FUNCTION_BLOCK PsdChuck EXTENDS ChuckBase
VAR_INPUT
	IoChuckPsd : IoChuckPsd;
END_VAR
VAR_OUTPUT
END_VAR
VAR
	{attribute 'OPC.UA.DA' := '0'}
	_config : PsdChuckConfig;
	
	{attribute 'OPC.UA.DA' := '0'}
	_deliverMessages : INT;
	
	WaferPresenceMsg : STRING(255);
	
	{attribute 'OPC.UA.DA' := '0'}
	_initDevice : BOOL;
	
	{attribute 'OPC.UA.DA' := '0'}
	_itemInit : INT;
	
	{attribute 'OPC.UA.DA' := '0'}
	_itemScheduler : INT;
	{attribute 'OPC.UA.DA' := '0'}
	_itemRaisedProperties : INT;
	{attribute 'OPC.UA.DA' := '0'}
	_pulseGenerator : TON;
	
	{region 'Commands'}
		
	{attribute 'OPC.UA.DA' := '0'}			  		   
	_raisePropertiesCmd : BOOL;
			
	{endregion}	
		
	{attribute 'OPC.UA.DA' := '0'}
	message : STRING;
	{attribute 'OPC.UA.DA' := '0'}
	_waferPresenceSensorCounter : UINT;
		 
END_VAR

SUPER^();

// Init device
InitDevice(); 

// Deliver messages
CASE _deliverMessages OF		
	EFeedbackMsgPsdChuck.WaferPresenceMsg :
		WaferPresenceMsg := message;		
END_CASE
	
_deliverMessages := 0;

// Commands	
RaisePropertiesChanged(_raisePropertiesCmd);

IF (NOT _raisePropertiesCmd) THEN
	MessageScheduler();
END_IF

METHOD FB_init : BOOL
VAR_INPUT
	bInitRetains : BOOL; // if TRUE, the retain variables are initialized (warm start / cold start)
	bInCopyCode : BOOL;  // if TRUE, the instance afterwards gets moved into the copy code (online change)
	Config : PsdChuckConfig;
END_VAR
IF Config.IsEnabled THEN
	_config := Config;
	
	SUPER^._chuckConfig.Name := Config.Name;
	SUPER^._chuckConfig.DeviceID := Config.DeviceID;
	SUPER^._chuckConfig.IsEnabled := Config.IsEnabled;
	SUPER^._chuckConfig.LogLevel := Config.LogLevel;
	
	SUPER^.Name := Config.Name;
	SUPER^.DeviceID := Config.DeviceID;
	
	THIS^.Family := DeviceFamily.Chuck;

	THIS^.SetReady();
	_Logger.Information(_message.Reset().Append('Init ').
							Append('{').Append(TO_STRING(THIS^.Family)).Append('} - ').
							Append('{').Append(TO_STRING(THIS^.Name)).Append('} - ').
							Append('Status : ').Append(TO_STRING(THIS^.Status)).
							ToString());										 
END_IF
END_METHOD

METHOD InitDevice
VAR_INPUT
END_VAR
IF NOT _initDevice THEN			
	_logger.Information(_message.Reset().
								Append(_config.Name).
								Append(' - init device').ToString());		
								
	_initDevice := TRUE;
END_IF
END_METHOD

METHOD MessageScheduler
VAR_INPUT
END_VAR
IF _pulseGenerator.Q THEN
	_pulseGenerator(IN := FALSE, PT := T#10MS);
		
	CASE _itemScheduler OF	
		0:	WaferPresenceMsg := ' ';
			_itemScheduler := 1;
	
		1:	ReadWaferPresence();
			_itemScheduler := 0;		
									
	END_CASE
ELSE
	_pulseGenerator(IN := TRUE, PT := T#100MS);	
END_IF
END_METHOD

{attribute 'TcRpcEnable' := '1'}
METHOD RaisePropertiesChanged
VAR_INPUT
	Execute : BOOL;
END_VAR
VAR	
	waferPresence : STRING;
	diameter : STRING;
END_VAR
IF Execute THEN		
	_raisePropertiesCmd := TRUE;	
	
	IF _pulseGenerator.Q THEN
		_pulseGenerator(IN := FALSE, PT := T#10MS);
		
		CASE _itemRaisedProperties OF		
			0:  diameter := TO_STRING(_config.WaferPresenceSensor[_waferPresenceSensorCounter].Diameter);
				WaferPresenceMsg := CONCAT(CONCAT(diameter, ';'), INT_TO_STRING(EMaterialPresence.Unknown));
				_itemRaisedProperties := 10;
				
			10: _logger.Information(_message.Reset().Append(_config.Name).Append(' - RaisePropertiesChanged').ToString());
				_raisePropertiesCmd := FALSE;
				_itemRaisedProperties := 0;		
		END_CASE	
	ELSE
		_pulseGenerator(IN := TRUE, PT := T#100MS);	
	END_IF		
END_IF
END_METHOD

METHOD ReadWaferPresence
VAR_INPUT
END_VAR
VAR	
	waferPresence : STRING;
	diameter : STRING;
END_VAR
_deliverMessages := EFeedbackMsgPsdChuck.WaferPresenceMsg;

IF _waferPresenceSensorCounter < Const.PSD_NUMBER_WAFER_PRESENCE_SENSORS - 1 THEN
	_waferPresenceSensorCounter := _waferPresenceSensorCounter + 1;
ELSE
	_waferPresenceSensorCounter := 0;
END_IF

diameter := TO_STRING(_config.WaferPresenceSensor[_waferPresenceSensorCounter].Diameter);
IF _config.WaferPresenceSensor[_waferPresenceSensorCounter].InputWaferPresence THEN
	waferPresence := INT_TO_STRING(EMaterialPresence.Present);
ELSE
	waferPresence := INT_TO_STRING(EMaterialPresence.NotPresent);		
END_IF

message := CONCAT(CONCAT(diameter, ';'), waferPresence);
END_METHOD

END_FUNCTION_BLOCK

(* stored: Version 1.1.0.1, ProductVersion 3.1.4024.12
   POU PsdChuck: Id {56b8a35a-5f6b-4f98-a4b9-2397fb2dd689}, SpecialFunc None
   Folder Commands: Id {61621eb1-94b0-4b03-9271-888005c2934d}
   Method FB_init: Id {f52019d8-75dd-4c64-a8c6-2e2af8e7e757}
   Method InitDevice: Id {d5df8234-9ecd-4f13-964f-343bf91ec072}
   Method MessageScheduler: Id {fa8a3e0e-a3b5-415c-91d2-ed9db904a976}
   Method RaisePropertiesChanged: Id {a25de0c6-b075-4ea7-bce3-1d10e903b33b}
   Method ReadWaferPresence: Id {0c159c27-7c95-47e5-8b5f-235439f0cf2c} *)
